RoboDK station: Robot unmerged table.rdk

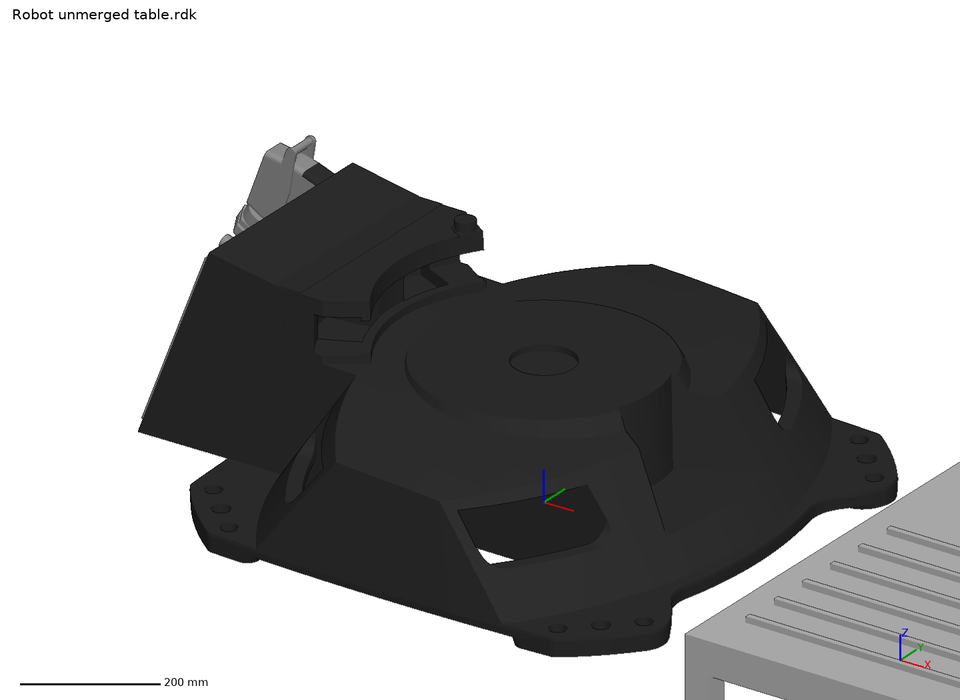
[picture v0: the station drawn from its stored meshes, robots at their saved joint values, targets as dots, program paths as lines]
Station Robot unmerged table (saved by RoboDK 5.2.3). Poses are relative to the parent item; angles as X-Y-Z fixed-axis rotations.
  - frame KUKA KR 210 R2700 extra Base at (0, 1000, 0) mm
    - robot KUKA KR 210 R2700 extra: 6 axes, payload 210 kg, reach 2696 mm, repeatability 0.06 mm, weight 1068 kg
        joint limits [-185, -140, -120, -350, -125, -350] to [185, -5, 155, 350, 125, 350]; home [0, -90, 90, 0, 0, 0]; saved at [0, -132.562, 125.475, 0, 7.088, 0]
      - tool Spindle, TCP at (278.6, 0, 88) mm, rotated rx 0 ry 90 rz 0 deg, size 85 x 346.5 x 128 mm
  - object FrameLeg at (1700, 300, 400) mm, rotated rx 0 ry 0 rz 90 deg, size 40 x 40 x 400 mm, geometry from FrameLeg.stl
  - object FramePLate at (1700, 300, 400) mm, rotated rx 0 ry 0 rz 90 deg, size 1810 x 1600 x 25 mm, geometry from FramePLate.stl
  - object FrameTop at (1700, 300, 400) mm, rotated rx 0 ry 0 rz 90 deg, size 1820 x 1605 x 60 mm, geometry from FrameTop.stl
  - object FrameSupport at (1700, 300, 400) mm, rotated rx 0 ry 0 rz 90 deg, size 20 x 1520 x 40 mm, geometry from FrameSupport.stl
  - object FrameSupport at (1700, -140, 400) mm, rotated rx 0 ry 0 rz 90 deg, size 20 x 1520 x 40 mm, geometry from FrameSupport.stl
  - object FrameSupport at (1700, -580, 400) mm, rotated rx 0 ry 0 rz 90 deg, size 20 x 1520 x 40 mm, geometry from FrameSupport.stl
  - object FrameLeg at (135, 300, 400) mm, rotated rx 0 ry 0 rz 90 deg, size 40 x 40 x 400 mm, geometry from FrameLeg.stl
  - object FrameLeg at (135, 2070, 400) mm, rotated rx 0 ry 0 rz 90 deg, size 40 x 40 x 400 mm, geometry from FrameLeg.stl
  - object FrameLeg at (1700, 2070, 400) mm, rotated rx 0 ry 0 rz 90 deg, size 40 x 40 x 400 mm, geometry from FrameLeg.stl
